// TIA Portal V20 export
DATA_BLOCK "DB_AsiSetpoint"   // DB24
// stored: Access Published, MemoryReserve 100, Namespace EmptyLine
   VAR
      Line : Struct
         EmptyLine : Struct
            DirChange : Struct
               Conveyor : Array[_.minEmptyLine.._.maxEmptyLine] of Bool;
            END_STRUCT;
            Speed : Struct
               Conveyor : Array[_.minEmptyLine.._.maxEmptyLine] of Bool;
            END_STRUCT;
         END_STRUCT;
      END_STRUCT;
   END_VAR
BEGIN
END_DATA_BLOCK
